TYPE U_OUT_IO_Translate :
UNION
	bArray :	ARRAY[1..32] OF BOOL;
	_Label :		OUTPUT_LABELS;
END_UNION
END_TYPE

(* stored: Version 1.1.0.1, ProductVersion 3.1.4024.10
   DUT U_OUT_IO_Translate: Id {2be7334c-18e8-47e6-91e2-0b0f98c4eb5e} *)
